(* CODESYS project BendingMachine.project
   Title: BendingMachine
   Version: 0.0.0.0
   Author: Enes

Project tree, tasks and I/O mapping:
  MyController : TM241C24T/U, Schneider Electric, order no. TM241C24T/U, version 4.0.6.18
    application Application
      task MAST (cyclic, interval 20 ms, priority 15, watchdog 100 ms x 1) calls POU
      global variables GVL
      program POU [LD]
      FunctionBlocks/
        function block Motor_Control [LD]
    DI : Digital Inputs, Schneider Electric, version 4.0.6.18
        input  iwDI_IW0 : WORD  // IW0
        input  ibDI_IB1 : BYTE  // IB1
    DQ : Digital Outputs, Schneider Electric, version 4.0.6.18
        settings: Outputs Usage = 3
        output qwDQ_QW0 : WORD  // QW0
        output qbDQ_QB1 : BYTE  // QB1
    Counters : Counters, Schneider Electric, version 4.0.6.18
    Pulse_Generators : Pulse Generators, Schneider Electric, version 4.0.6.18
        settings: Instance name = 'Axis_1'; B output History = 'old=-1 new=1'; A output History = 'old=-1 new=0'; Temporary Instance name = 'Axis_1'
    Cartridge_1 : Cartridge, Schneider Electric, version 4.0.6.18
    IO_Bus : IO bus - TM3, Schneider Electric, version 4.0.6.18
    COM_Bus : COM bus, Schneider Electric, version 4.0.6.18
    Serial_Line_1 : Serial line, Schneider Electric, version 4.0.6.18
      SoMachine_Network_Manager : SoMachine-Network Manager, Schneider Electric, version 4.0.0.2
    Serial_Line_2 : Serial line, Schneider Electric, version 4.0.6.18
      Modbus_Manager : Modbus Manager, Schneider Electric, version 4.0.0.2
*)

// MyController/Application/GVL
VAR_GLOBAL
	Power_En: BOOL;
	Stop_En: BOOL;
	Reset_En: BOOL;
	Home_En: BOOL;
	MoveToBending_En: BOOL;
	MoveToHome_En: BOOL;
END_VAR

// MyController/Application/POU
PROGRAM POU
VAR
	Motor_Control_FB: Motor_Control;
	Sensor_Detected: BOOL;
	BendingMachine: BOOL;
	Timer_1: TON;
	Timer_2: TON;
	Timer_3: TON;
	CTU_0: CTU;
	StopForBending: BOOL;
	Start_Button: BOOL;
	Start: BOOL;
	Stop_Button: BOOL;
	Resume_Button: BOOL;
	AfterBending: BOOL;
	GoHome: BOOL;
	StartSystem: BOOL;
	ResumeSystem_1: BOOL;
	ResumeSystem_2: BOOL;
END_VAR
VAR // added by the converter: edge detectors and wires of the graphical bodies
    _w1, _w2, _w3 : BOOL;
    _rt1 : R_TRIG;
END_VAR

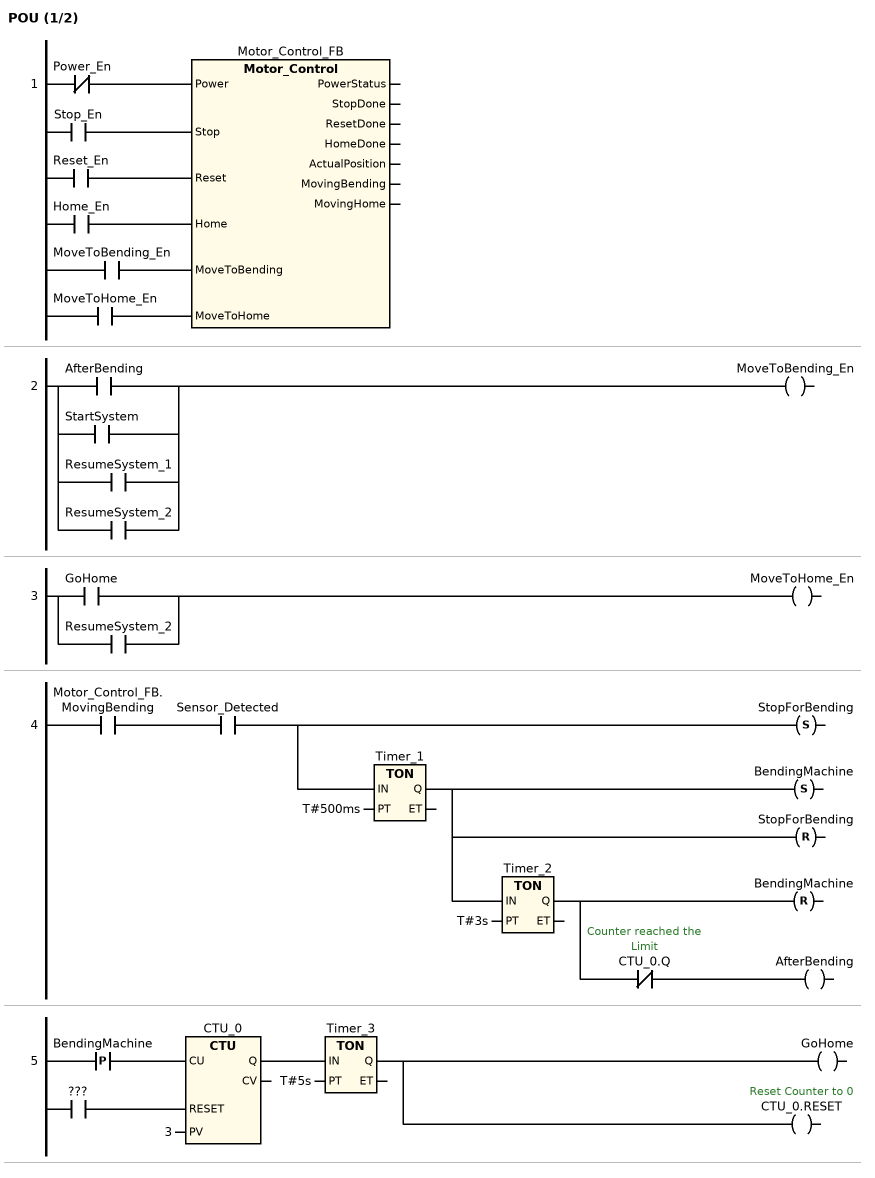
// NETWORK 1
Motor_Control_FB(
    Power := NOT Power_En,
    Stop := Stop_En,
    Reset := Reset_En,
    Home := Home_En,
    MoveToBending := MoveToBending_En,
    MoveToHome := MoveToHome_En); // Motor_Control

// NETWORK 2
MoveToBending_En := AfterBending OR StartSystem OR ResumeSystem_1 OR ResumeSystem_2;

// NETWORK 3
MoveToHome_En := GoHome OR ResumeSystem_2;

// NETWORK 4
//   CTU_0.Q: Counter reached the Limit
_w1 := Motor_Control_FB.MovingBending AND Sensor_Detected;
StopForBending S= _w1;
Timer_1(IN := _w1, PT := T#500ms); // TON
BendingMachine S= Timer_1.Q;
StopForBending R= Timer_1.Q;
Timer_2(IN := Timer_1.Q, PT := T#3s); // TON
BendingMachine R= Timer_2.Q;
AfterBending := Timer_2.Q AND NOT CTU_0.Q;

// NETWORK 5
//   CTU_0.RESET: Reset Counter to 0
_rt1(CLK := BendingMachine);
CTU_0(CU := _rt1.Q, PV := 3); // CTU
Timer_3(IN := CTU_0.Q, PT := T#5s); // TON
GoHome := Timer_3.Q;
CTU_0.RESET := Timer_3.Q;

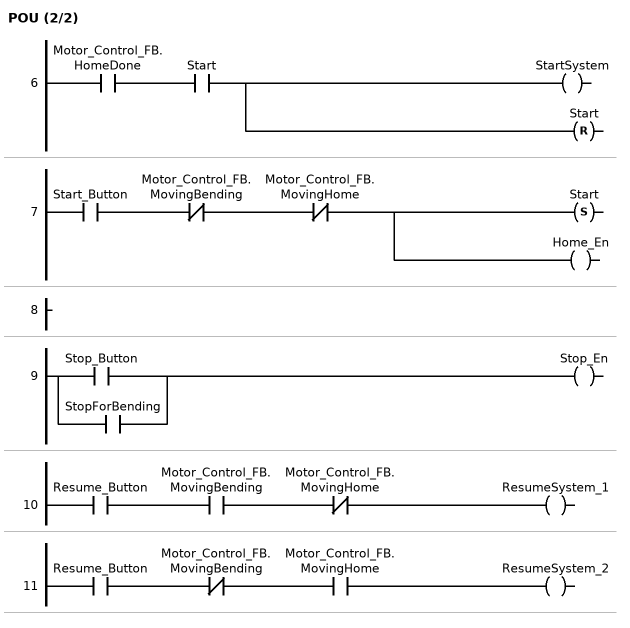
// NETWORK 6
_w2 := Motor_Control_FB.HomeDone AND Start;
StartSystem := _w2;
Start R= _w2;

// NETWORK 7
_w3 := Start_Button AND NOT Motor_Control_FB.MovingBending AND NOT Motor_Control_FB.MovingHome;
Start S= _w3;
Home_En := _w3;

// NETWORK 8

// NETWORK 9
Stop_En := Stop_Button OR StopForBending;

// NETWORK 10
ResumeSystem_1 := Resume_Button AND Motor_Control_FB.MovingBending AND NOT Motor_Control_FB.MovingHome;

// NETWORK 11
ResumeSystem_2 := Resume_Button AND NOT Motor_Control_FB.MovingBending AND Motor_Control_FB.MovingHome;

END_PROGRAM

// MyController/Application/FunctionBlocks/Motor_Control
FUNCTION_BLOCK Motor_Control
VAR_INPUT
	Power: BOOL;
	Stop: BOOL;
	Reset: BOOL;
	Home: BOOL;
	MoveToBending: BOOL;
	MoveToHome: BOOL;
END_VAR
VAR_OUTPUT
	PowerStatus: BOOL;
	StopDone: BOOL;
	ResetDone: BOOL;
	HomeDone: BOOL;
	ActualPosition: DINT;
	MovingBending: BOOL;
	MovingHome: BOOL;
END_VAR
VAR
	MC_Power: MC_Power_PTO;
	MC_Stop: MC_Stop_PTO;
	MC_Reset: MC_Reset_PTO;
	MC_Home: MC_Home_PTO;
	MC_MoveAbsolute_Forward: MC_MoveAbsolute_PTO;
	MC_MoveAbsolute_Reverse: MC_MoveAbsolute_PTO;
	MC_ReadActualPosition: MC_ReadActualPosition_PTO;
	Forward: BOOL;
	Reverse: BOOL;
END_VAR
VAR // added by the converter: edge detectors and wires of the graphical bodies
    _rt1, _rt2 : R_TRIG;
END_VAR

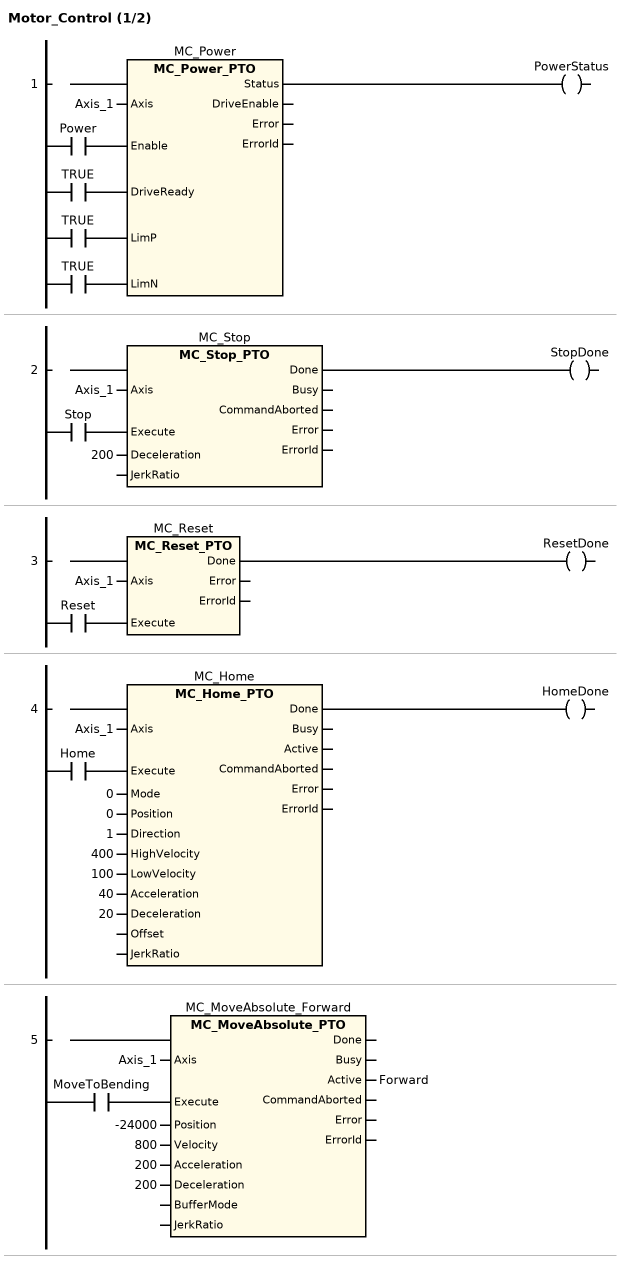
// NETWORK 1
MC_Power(Axis := Axis_1, Enable := Power, DriveReady := TRUE, LimP := TRUE, LimN := TRUE); // MC_Power_PTO
PowerStatus := MC_Power.Status;

// NETWORK 2
MC_Stop(Axis := Axis_1, Execute := Stop, Deceleration := 200); // MC_Stop_PTO
StopDone := MC_Stop.Done;

// NETWORK 3
MC_Reset(Axis := Axis_1, Execute := Reset); // MC_Reset_PTO
ResetDone := MC_Reset.Done;

// NETWORK 4
MC_Home(
    Axis := Axis_1,
    Execute := Home,
    Mode := 0,
    Position := 0,
    Direction := 1,
    HighVelocity := 400,
    LowVelocity := 100,
    Acceleration := 40,
    Deceleration := 20); // MC_Home_PTO
HomeDone := MC_Home.Done;

// NETWORK 5
MC_MoveAbsolute_Forward(
    Axis := Axis_1,
    Execute := MoveToBending,
    Position := -24000,
    Velocity := 800,
    Acceleration := 200,
    Deceleration := 200,
    Active => Forward); // MC_MoveAbsolute_PTO

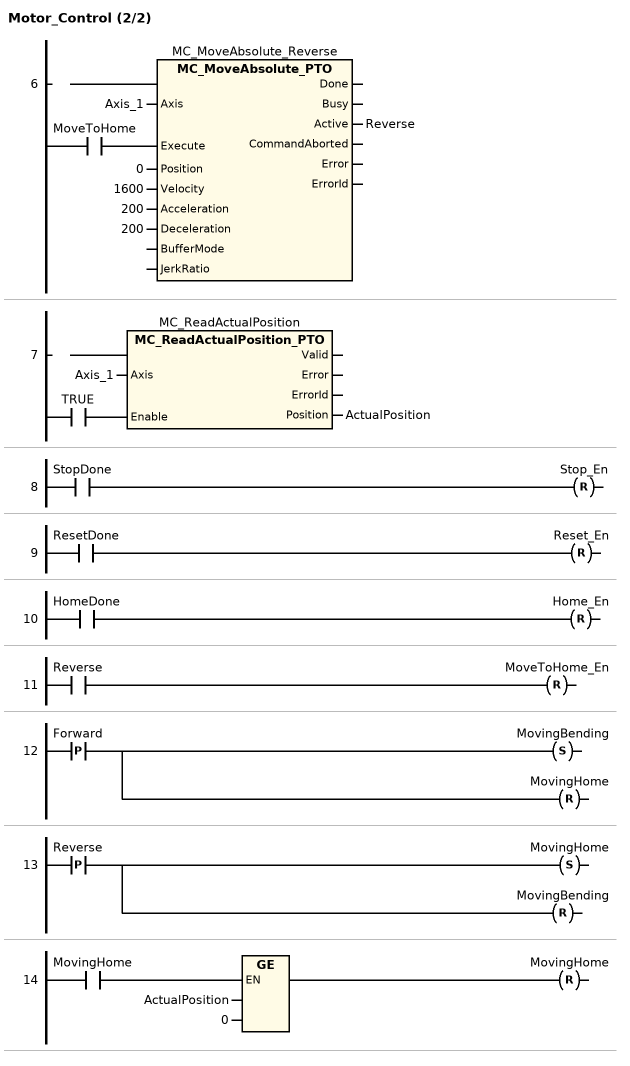
// NETWORK 6
MC_MoveAbsolute_Reverse(
    Axis := Axis_1,
    Execute := MoveToHome,
    Position := 0,
    Velocity := 1600,
    Acceleration := 200,
    Deceleration := 200,
    Active => Reverse); // MC_MoveAbsolute_PTO

// NETWORK 7
MC_ReadActualPosition(Axis := Axis_1, Enable := TRUE, Position => ActualPosition); // MC_ReadActualPosition_PTO

// NETWORK 8
Stop_En R= StopDone;

// NETWORK 9
Reset_En R= ResetDone;

// NETWORK 10
Home_En R= HomeDone;

// NETWORK 11
MoveToHome_En R= Reverse;

// NETWORK 12
_rt1(CLK := Forward);
MovingBending S= _rt1.Q;
MovingHome R= _rt1.Q;

// NETWORK 13
_rt2(CLK := Reverse);
MovingHome S= _rt2.Q;
MovingBending R= _rt2.Q;

// NETWORK 14
MovingHome R= MovingHome AND ActualPosition >= 0;

END_FUNCTION_BLOCK
